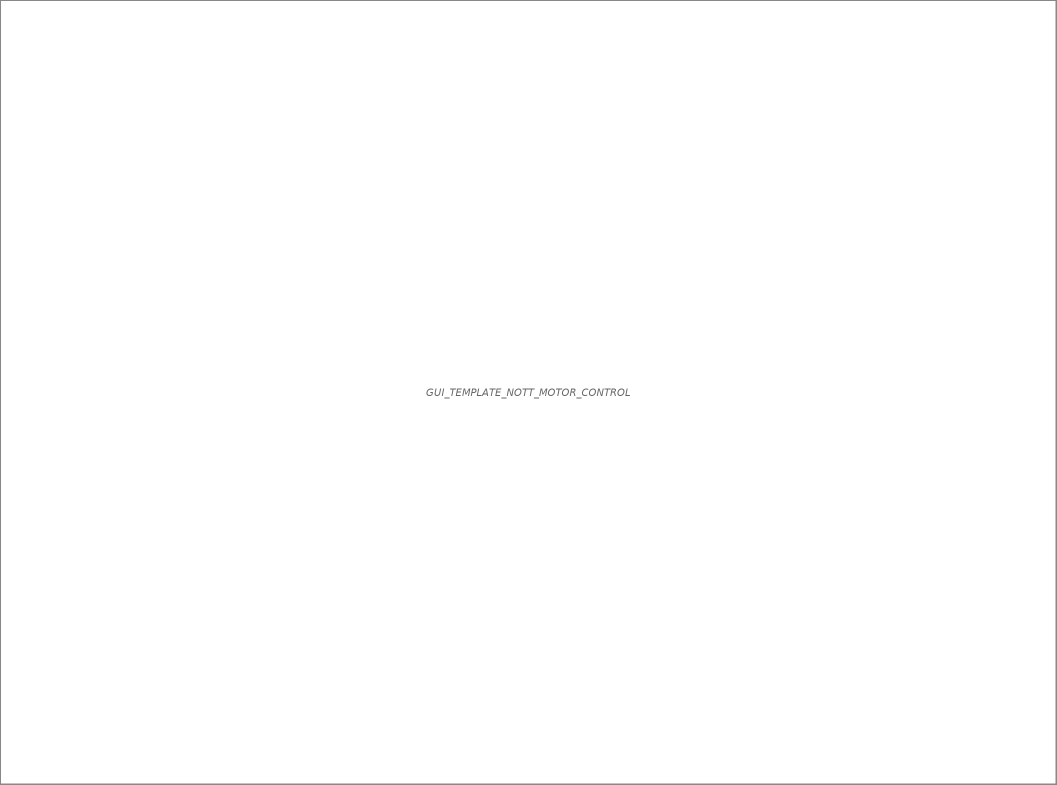
VISUALIZATION GUI_TEMPLATE_MOTOR  // 1057x785
VAR_IN_OUT
	m_Instance:	FB_NOTT_MOTOR;
END_VAR
VAR
	m_lrOffSet : LREAL := 0;
END_VAR
    TabControl (0,0 1057x785)
        shows GUI_TEMPLATE_NOTT_MOTOR_CONTROL(m_Instance := m_Instance)
        shows GUI_TEMPLATE_NOTT_MOTOR_CONFIG(m_Instance := m_Instance)
        [0]: TabTitle=Control
        [1]: TabTitle=Config
END_VISUALIZATION

(* stored: Version 1.1.0.1, ProductVersion 3.1.4024.14
   Visu GUI_TEMPLATE_MOTOR: Id {81aa027d-a672-455f-898b-33573355b743} *)
